TEXTLIST TL_ModeSwitchState_1
  0 = 'Auto'
  1 = 'Manual'
   = ''
END_TEXTLIST

(* stored: Version 1.1.0.1, ProductVersion 3.1.4024.12
   TextList TL_ModeSwitchState_1: Id {57786b28-7f19-457c-af93-163f552f5f8b} *)
